FUNCTION_BLOCK FB_MotionStageSim_Test EXTENDS TcUnit.FB_TestSuite
VAR
    Expected: BOOL := True;
    Actual: BOOL;
END_VAR

TEST('FB_MotionStageSim_Test Dummy Test');
AssertEquals(Expected := Expected,
             Actual := Actual,
             Message := 'Error Message');
TEST_FINISHED();

END_FUNCTION_BLOCK

(* stored: Version 1.1.0.1, ProductVersion 3.1.4022.18
   POU FB_MotionStageSim_Test: Id {438b9682-8d81-4225-ac01-d9e819d04a63}, SpecialFunc None *)
